TYPE ST_InfeedCommand :
	STRUCT
		StartConveyor : BOOL;
		StopConveyor  : BOOL;
	END_STRUCT
END_TYPE

(* stored: Version 1.1.0.1, ProductVersion 3.1.4024.12
   DUT ST_InfeedCommand: Id {480a2c3d-4f6c-42ee-9693-75f364808c87} *)
